FUNCTION_BLOCK BYPASS_AX_AX (* Bypass FB *)
  (* Standard: 61499-2 *)
  (* Version 1.0, 2026-05-07, franz *)
  PACKAGE logiBUS::signalprocessing::bypass;
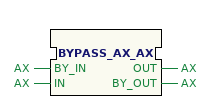
  SOCKETS
    BY_IN : adapter::types::unidirectional::AX; (* Bypass in *)
    IN : adapter::types::unidirectional::AX; (* Signal Input *)
  END_SOCKETS
  PLUGS
    OUT : adapter::types::unidirectional::AX; (* Signal Output *)
    BY_OUT : adapter::types::unidirectional::AX; (* Bypass out *)
  END_PLUGS
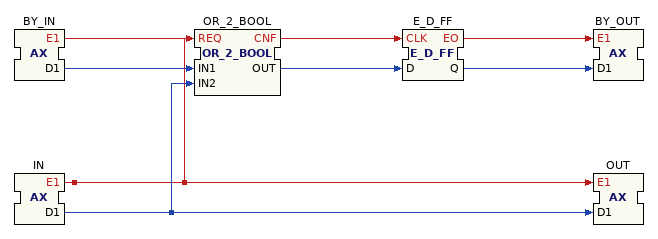
  FBS
    OR_2_BOOL : iec61131::booleanOperators::OR_2_BOOL;
    E_D_FF : iec61499::events::E_D_FF;
  END_FBS
  EVENT_CONNECTIONS
    IN.E1 TO OUT.E1;
    BY_IN.E1 TO OR_2_BOOL.REQ;
    IN.E1 TO OR_2_BOOL.REQ;
    OR_2_BOOL.CNF TO E_D_FF.CLK;
    E_D_FF.EO TO BY_OUT.E1;
  END_CONNECTIONS
  DATA_CONNECTIONS
    IN.D1 TO OUT.D1;
    BY_IN.D1 TO OR_2_BOOL.IN1;
    IN.D1 TO OR_2_BOOL.IN2;
    OR_2_BOOL.OUT TO E_D_FF.D;
    E_D_FF.Q TO BY_OUT.D1;
  END_CONNECTIONS
END_FUNCTION_BLOCK
